(* PLC project AufgSer3, Beckhoff Automation GmbH TwinCAT PLC Control 3.5.13.21 *)
(* stored: creationDateTime 2022-04-25T13:35:32.6922168, modificationDateTime 2022-04-25T13:35:32.6922168 *)

FUNCTION F_Square : REAL
VAR_INPUT
	ymin	: REAL;	// Minimalwert
	ymax	: REAL;	// Maximalwert
	yoff	: REAL; // offset
	w		: REAL; // Kreisfrequenz (rad/s)
	t		: REAL; // Time (s)
END_VAR
VAR
	sinRes	: REAL; // sine result
	squareRes: REAL;
END_VAR

            sinRes := SIN(w*t);

IF (sinRes > 0) THEN
	squareRes := ymin;
ELSE
	squareRes := ymax;
END_IF

F_Square := squareRes + yoff;
          
END_FUNCTION
